Staubli VAL3: PublicData.dtx

public bool bByPass[4]
public bool bSimulaiton
public jointRx jHome = {j1=-103.334484, j2=39.165058, j3=105.338631, j4=-0.126343, j5=35.633301, j6=76.948067}
public mdesc mFast = {accel=30, decel=30, rmax=600, tmax=200, leave=2, reach=2}
public mdesc mHome = {accel=20, decel=20, tmax=200, blend=cartesian, leave=5, reach=5}
public mdesc mMiddleFast = {accel=20, decel=20, tmax=150, blend=cartesian, leave=1, reach=1}
mdesc mNomSpeed
public mdesc mSlow = {accel=10, decel=19, rmax=100, tmax=50, blend=cartesian, leave=1, reach=1}
public num nBeltLife = 1000
public num nCompenCount = 0.001
public num nDelta
public num nSumCompen = 0.2
public string sCurrentPrd = "P1"
public string sPrd = "P1"
public string sProductList = "C2300"
public string sStartPrd = "P1"
public string sStatus = "stop"
